PROGRAM MAIN
VAR
END_VAR

END_PROGRAM

(* stored: Version 1.1.0.1
   POU MAIN: Id {08840ecc-cfd9-4914-96cc-57351a117aee} *)
